PROGRAM MAIN
VAR
	
END_VAR

//In Main we just run all our program for pick and place stack mashine. 
//As you can see we have 6 program and a HMI program for our mashine. 

P_1Start();
P_2PickUP();
P_3Pack();
P_4Packing();
P_5MovingToStack();
P_6Stack();
HMI();

END_PROGRAM

(* stored: Version 1.1.0.1, ProductVersion 3.1.4024.3
   POU MAIN: Id {7f7638e9-7a1d-4c26-91a2-7aeecf20f056}, SpecialFunc None *)
